// TIA Portal V20 export
DATA_BLOCK "ControlNodes"   // DB199
// stored: MemoryReserve 100, Namespace Unit1.Em3
   VAR
      em { ExternalWritable := 'False'} : "LAF_typeEmControlNode";
      cm { ExternalWritable := 'False'} : "Unit1.Em3.typeCmControlNode";
      citiMap : "LER_OEM_Data";
      webGuid { ExternalWritable := 'False'} : "Unit1.Em3.typeSequenceControlNode";
   END_VAR
   VAR RETAIN
      cmMasterVirtualAxis { ExternalWritable := 'False'} : "LBC_typeAxisControlNode";
      cmUnwinderVirtualAxis { ExternalWritable := 'False'} : "LBC_typeAxisControlNode";
      cmDancerRegulatorOnOff { ExternalWritable := 'False'} : "LBC_typeTwoWayActuatorControlNode";
      cmDancerSafetyPinIdlePosition { ExternalWritable := 'False'} : "LBC_typeDigitalSignalControlNode";
      cmLoadCellAnalogInput { ExternalWritable := 'False'} : "LBC_typeAnalogInputControlNode";
      cmDancerEncoderAnalogInput { ExternalWritable := 'False'} : "LBC_typeAnalogInputControlNode";
      cmDancerElectroPneumaticRegulatorAnalogOutput { ExternalWritable := 'False'} : "LBC_typeAnalogOutputControlNode";
      cmWebGuideEpc { ExternalWritable := 'False'} : "LER_typeCON600ControlNode";
   END_VAR
   VAR
      cmDancerRegulatorOutput { ExternalWritable := 'False'} : LReal;
   END_VAR
BEGIN
END_DATA_BLOCK
